{attribute addProperty BoxType "EPP1342-0001-0016"}
{attribute addProperty Id "InfoDataInfoData_192954DE162"}
{attribute addProperty CRC "395970889"}
{attribute addProperty SizeInBites "16"}
{attribute addProperty SizeInBytes "2"}
TYPE EPP1342_179A0949 :
STRUCT
	{attribute addProperty Name "InfoData"}
	InfoData : InfoData_192954DE;
END_STRUCT
END_TYPE

(* stored: Version 1.2.0.0, ProductVersion 3.1.4024.9
   DUT EPP1342_179A0949: Id {857c4962-9036-443f-b45d-d3677c1e19ae} *)
